PROGRAM PRG_10ms
VAR
	fbVirtualCOM							:SerialLineControlADS;
	fbComRec								:ReceiveData;
	fbComSend							:SendData;
	Delay									:TON;
	
	stCOMSerialConfig					:ComSerialConfig;	
	TXBuffer,RXBuffer					:ComBuffer;	
	aDataRec								:ARRAY[0..19] OF BYTE;
	aDataSend								:ARRAY[0..19] OF BYTE;
	bInit										:BOOL := TRUE;
END_VAR

stCOMSerialConfig.ComPort := 1;
stCOMSerialConfig.Baudrate := 9600;
stCOMSerialConfig.Parity := PARITY_EVEN;
stCOMSerialConfig.DataBits := 7;
stCOMSerialConfig.StopBits := STOPBITS_ONE;

fbVirtualCOM(
	Connect:= bInit, 
	SerialCfg:= stCOMSerialConfig, 
	NetId:= , 
	Timeout:= , 
	TxBuffer:= TXBuffer, 
	RxBuffer:= RXBuffer, 
	PortOpened=> , 
	Error=> , 
	ErrorID=> , 
	Busy=> , 
	TxBufCount=> , 
	RxBufCount=> );

Delay(IN:=NOT Delay.Q, PT := T#500MS);	
IF Delay.Q AND fbVirtualCOM.PortOpened THEN	
fbComSend(
	pSendData:= ADR(aDataSend), 
	Length:= SIZEOF(aDataSend), 
	Busy=> , 
	Error=> , 
	TXbuffer:= TXBuffer);	
END_IF
	
fbComRec(
	pPrefix:= , 
	LenPrefix:= , 
	pSuffix:= , 
	LenSuffix:= , 
	pReceiveData:= ADR(aDataRec), 
	SizeReceiveData:= SIZEOF(aDataRec), 
	Timeout:= , 
	Reset:= , 
	DataReceived=> , 
	busy=> , 
	Error=> , 
	RxTimeout=> , 
	LenReceiveData=> , 
	RXbuffer:= RXBuffer);

END_PROGRAM

(* stored: Version 1.1.0.1, ProductVersion 3.1.4024.9
   POU PRG_10ms: Id {db08171f-adc1-4570-8775-54830cad8d14}, SpecialFunc None *)
